PROGRAM PDODatenMotor
VAR
	StromPDOMotor1 AT%I* 		: INT;
	SpannungPDOMotor1 AT%I*		: UINT;
	StromPDOMotor2 AT%I* 		: INT;
	SpannungPDOMotor2 AT%I*	 	: UINT;
	StromPDOMotor3 AT%I* 		: INT;
	SpannungPDOMotor3 AT%I*		: UINT;
	
	StromPDOGreifer AT%I*		: INT;
	SpannungPDOGreifer AT%I*	: UINT;
END_VAR

(*	Strom und Spannung des Motors werden direkt per PDO-Mapping als Outputs gemappt
	Hier: nur Input Variablen definiert, um die Daten im Scope Server anzeigen zu lassen
*)

END_PROGRAM

(* stored: Version 1.1.0.1, ProductVersion 3.1.4022.3
   POU PDODatenMotor: Id {cb7a9b27-fcc7-4f64-af1c-7d4defbe2f79}, SpecialFunc None *)
